FUNCTION_BLOCK BoxLoader
VAR_INPUT
END_VAR
VAR_OUTPUT
END_VAR
VAR
END_VAR

END_FUNCTION_BLOCK

(* stored: Version 1.1.0.1, ProductVersion 3.1.4024.2
   POU BoxLoader: Id {8c060388-5aea-4670-8177-a59a4980b218}, SpecialFunc None *)
